// TIA Portal V20 export
TYPE "IO_CONTVLV"
   STRUCT
      IN { ExternalAccessible := 'False'; ExternalVisible := 'False'; ExternalWritable := 'False'} : Struct
         OpenFb : Bool;
         ClosedFb : Bool;
         PositionFb : Real;
         Fault : Bool;
      END_STRUCT;
      OUT { ExternalAccessible := 'False'; ExternalVisible := 'False'; ExternalWritable := 'False'} : Struct
         OpenCmd : Bool;
         CloseCmd : Bool;
         PositionCmd : Real;
      END_STRUCT;
   END_STRUCT;
END_TYPE
